FUNCTION MultiplyMatrix3 : ARRAY[0..2, 0..2] OF LREAL
VAR_INPUT
	matrix : ARRAY[0..2,0..2] OF LREAL;
	multiplier : LREAL;
END_VAR

VAR
	i, j : INT;
END_VAR

FOR i := 0 TO 2 DO
	FOR j := 0 TO 2 DO
		MultiplyMatrix3[i, j] := matrix[i, j] * multiplier;
	END_FOR;
END_FOR

END_FUNCTION

(* stored: Version 1.1.0.1, ProductVersion 3.1.4024.11
   POU MultiplyMatrix3: Id {fdd6595b-fa60-401c-a9b6-d71a39c93ebd}, SpecialFunc None *)
